(* CODESYS project SingleElevator_ancestor.project

Project tree, tasks and I/O mapping:
  Device : CODESYS Control Win V3, 3S - Smart Software Solutions GmbH, version 3.5.15.40
    application Application
      libraries: Standard, * (System)
      task MainTask (cyclic, interval 50 ms, priority 1) calls Simulation, GA_collector, Policy
      task VISU_TASK (cyclic, interval 100 ms, priority 31) calls VisuElems.Visu_Prg
      global variables GVL
      visualisation Visualization
      program Simulation [ST]
      GAs/
        function block Door_module [SFC]: ready_active, busy_active, op_complete_active, reset_done_active
        function block Dir_Vel_module [SFC]: go_fast_active, op_complete_active, reset_done_active, busy_active, ready_active, go_slow_active, stop_active
        function block Homing_Limit_module [SFC]: op_complete_active, reset_done_active, busy_active, ready_active, closing_doors_exit, closing_doors_active, slow_d_active, slow_u_active, opening_doors_active, opening_doors_exit, slow_u_top_active, slow_d_top_active, slow_d_exit, slow_u_exit, slow_u_top_exit, slow_d_top_exit, slow_d_bot_exit, slow_d_bot_exit_0, slow_u_bot_active, slow_d_bot_active, stop_h_active, stop_h_exit
        function block Calls_module [SFC]: Busy_active, Ready_active, op_complete_active, reset_done_active, save_up_active, Init_active, save_down_active, compose_array_up_active, compose_array_down_active
        function block Lights_module [SFC]: Ready_active, all_lights_active, Busy_active, save_call_active, save_call_exit
        function block Serve_call_module [SFC]: Ready_active, Busy_active, close_door_exit, slow_d_active, slow_d_exit, close_door_active, slow_u_active, fast_u_active, slow_u_land_active, Stop_active, Open_Doors_active, slow_u_exit, fast_u_exit, slow_u_land_exit, Stop_u_exit, Open_Doors_exit, fast_d_active, slow_d_land_active, Stop_d_active, fast_d_exit, slow_d_land_exit, Stop_d_exit, cancel_call_active, cancel_call_down_active, cancel_call_up_exit, cancel_call_down_exit
      program GA_collector [FBD]
      program Policy [SFC]: homing_active, homing_exit, wait_for_call_active
  text list GlobalTextList
*)

// Device/Application/GVL
//{attribute 'qualified_only'}
VAR_GLOBAL
(* Elevator managing variables*)
	Open: BOOL;				(* Sensor: the door is fully open*)
	Closed: BOOL;			(* Sensor: the door is fully closed*)
	LimitDown: BOOL;		(* Sensor: lower limit sensor, if TRUE the lift has reached the lower limit*)
	LimitUp: BOOL;			(* Sensor: upper limit sensor, if TRUE the lift has reached the upper limit*)
	DeckSensor: BOOL;		(* Sensor: if TRUE the cab is in proximity of a deck*)
	RampSensor: BOOL;		(* Sensor: if TRUE the cab is in proximity of a ramp*)
	Presence :BOOL; 		(* Sensor: if TRUE something blocks the door photocell*)
	Emergency: BOOL;		(* Input: if TRUE the emergency button has been pressed*)

	Closing: BOOL;			(* Actuator: if TRUE the door starts closing*)
	Opening: BOOL;			(* Actuator: the door starts opening*)
	Motor_on: BOOL;			(* Actuator: if TRUE the lift pulley motor start moving*)
	Up: BOOL;				(* Actuator parameter: if TRUE the lift moves upward, downward otherwise*)
	Vel: BOOL;				(* Actuator parameter: motor speed, if TRUE high speed, low speed otherwise*)
	

	Current: INT;  			(* Visualization: variable used to storage the current deck*)
    Destination: INT;		(* Visualization: variable used to storage the the destination deck*)
	EmergencyVis: BOOL; 	(* Visualization: if TRUE the emergency light is turned on*)

	
	
	
	
	
	InitialDeck: INT := 1;	(* Only for simulation: variable used to define the initial deck*)
	InitCycle: BOOL := FALSE;(* Only for simulation: used to execute the instruction at the first cycle*)
	Height: INT;			(* Only for simulation: elevator height*)
	DeckRest: INT;        	(* Only for simulation: division rest for generating deck sensor*)
	Memory: INT;
	RampRest: INT;			(* Only for simulation: division rest for generating the ramp position*)
	MemoryR: INT;
	Door: INT;				(* Only for simulation: to visualize the closing of the door*)
	Displacement: INT;		(* Only for simulation: lift displacement, dependent on the motor speed*)

 (*Inputs: internal panel variables*)
	PG: BOOL;
	P1: BOOL;
	P2: BOOL;
	P3: BOOL;
	P4: BOOL;
	P5: BOOL;
	P6: BOOL;
	P7: BOOL;

(*Visualization: internal panel variables used to turn on the LED*)
	PGVis: BOOL;
	P1Vis: BOOL;
	P2Vis: BOOL;
	P3Vis: BOOL;
	P4Vis: BOOL;
	P5Vis: BOOL;
	P6Vis: BOOL;
	P7Vis: BOOL;

(*Inputs: external panel variables*)
	UpDeckG: BOOL;
	UpDeck1: BOOL;
	UpDeck2: BOOL;
	UpDeck3: BOOL;
	UpDeck4: BOOL;
	UpDeck5: BOOL;
	UpDeck6: BOOL;
	DownDeck7: BOOL;
	DownDeck6: BOOL;
	DownDeck5: BOOL;
	DownDeck4: BOOL;
	DownDeck3: BOOL;
	DownDeck2: BOOL;
	DownDeck1: BOOL;

(*Visualization: external panel variables used to turn on the LED*)
	UpDeckGVis: BOOL;
	UpDeck1Vis: BOOL;
	UpDeck2Vis: BOOL;
	UpDeck3Vis: BOOL;
	UpDeck4Vis: BOOL;
	UpDeck5Vis: BOOL;
	UpDeck6Vis: BOOL;
	DownDeck7Vis: BOOL;
	DownDeck6Vis: BOOL;
	DownDeck5Vis: BOOL;
	DownDeck4Vis: BOOL;
	DownDeck3Vis: BOOL;
	DownDeck2Vis: BOOL;
	DownDeck1Vis: BOOL;

(*Only for simulation: variables used to simulate the fault on deck sensor*)
	SensorG: BOOL;				(* if TRUE the magnetic information for deck G is lost and the deck sensor cannot become TRUE*)
	Sensor1: BOOL;				(* if TRUE the magnetic information for deck 1 is lost and the deck sensor cannot become TRUE*)
	Sensor2: BOOL;
	Sensor3: BOOL;
	Sensor4: BOOL;
	Sensor5: BOOL;
	Sensor6: BOOL;
	Sensor7: BOOL;
	FaultSensorAlarm: BOOL; 	(* Visulaization: if TRUE alerts the user of a deck sensor fault*)

(*Only for simulation: variables used to simulate the fault on ramp sensor*)
	RampGUp: BOOL;
	Ramp1Down: BOOL;
	Ramp1Up:BOOL;
	Ramp2Down: BOOL;
	Ramp2Up:BOOL;
	Ramp3Down: BOOL;
	Ramp3Up:BOOL;
	Ramp4Down: BOOL;
	Ramp4Up:BOOL;
	Ramp5Down: BOOL;
	Ramp5Up:BOOL;
	Ramp6Down: BOOL;
	Ramp6Up:BOOL;
	Ramp7Down: BOOL;
	FaultRampAlarm: BOOL; 		(* Visulaization: if TRUE alerts the user of a ramp sensor fault*)
	SensorGOK: BOOL;
	Sensor1OK: BOOL;
	Sensor2OK: BOOL;
	Sensor6OK: BOOL;
	Sensor3OK: BOOL;
	Sensor4OK: BOOL;
	Sensor5OK: BOOL;
	Sensor7OK: BOOL;
	RampGUpOK: BOOL;
	Ramp1DownOK: BOOL;
	Ramp1UpOK: BOOL;
	Ramp2DownOK: BOOL;
	Ramp2UpOK: BOOL;
	Ramp3DownOK: BOOL;
	Ramp3UpOK: BOOL;
	Ramp4DownOK: BOOL;
	Ramp4UpOK: BOOL;
	Ramp5DownOK: BOOL;
	Ramp5UpOK: BOOL;
	Ramp6DownOK: BOOL;
	Ramp6UpOK: BOOL;
	Ramp7DownOK: BOOL;
	Ramp7UpOK: BOOL;
	//var aggiunte da me
	array_prio_up_onfly: ARRAY[0..7] OF INT;
	array_dest_up_onfly: ARRAY[0..7] OF INT;
	array_prio_up_stored: ARRAY[0..7] OF INT;
	array_dest_up_stored: ARRAY[0..7] OF INT;
	
	array_prio_down_onfly: ARRAY[0..7] OF INT;
	array_dest_down_onfly: ARRAY[0..7] OF INT;
	array_prio_down_stored: ARRAY[0..7] OF INT;
	array_dest_down_stored: ARRAY[0..7] OF INT;
	
	same_floor: BOOL; //flag di calls_module per la policy
	up_flag: BOOL; //
	RampSensor_target: BOOL;
	
	//Istanze dei GA
	door_module_0: Door_module;
	Dir_Vel_module_0: Dir_Vel_module;
	Homing_Limit_module_0: Homing_Limit_module;
	Lights_module_0: Lights_module;
	Calls_module_0: Calls_module;
	Serve_call_module_0: Serve_call_module;
	

END_VAR

// Device/Application/Simulation
PROGRAM Simulation
VAR
END_VAR

(* Initial position of the cab inside the hoistway. It is executed only at the first cycle.  *)
IF NOT GVL.InitCycle THEN
			GVL.InitCycle := TRUE ;
			GVL.Height := 20 * GVL.InitialDeck;
		    GVL.Door := 0;
			GVL.Current := GVL.Height / 20;
END_IF;

(* Elevator management, these instructions are executed each cycle time*)

(* Elevator door control. *)
IF GVL.Closing THEN
	GVL.Door := GVL.Door + 1;		(*Closing door management*)
	GVL.Open := FALSE;
END_IF

IF GVL.Door >= 60 THEN						(* Closed door limit*)
	GVL.Closed := TRUE;
END_IF

IF GVL.Opening THEN
	GVL.Door := GVL.Door - 1; 	(* Opening door management*)
	GVL.Closed := FALSE;
END_IF

IF GVL.Door <= 0 THEN							(* Open door limit*)
	GVL.Open := TRUE;
END_IF


(* Maximum and minimum management in the door simulation*)
IF GVL.Door < 0 THEN
	 GVL.Door := 0;
END_IF

IF GVL.Door > 60 THEN
	GVL.Door := 60;
END_IF


(* Control of the cab position inside the hostway. *)
(* Displacement definition for graphic visualization*)
IF GVL.Vel THEN 
	GVL.Displacement := 2;
ELSE 
	GVL.Displacement := 1;
END_IF


(* Height modification relying on direction and speed*)
IF GVL.Motor_on AND GVL.Up THEN
	GVL.Height := GVL.Height + GVL.Displacement;
	GVL.LimitDown := FALSE;
END_IF

IF GVL.Motor_on AND NOT GVL.Up THEN
	GVL.Height := GVL.Height - GVL.Displacement;
	GVL.LimitUp := FALSE;
END_IF


(* Limits for visualization*)
IF GVL.Height < -20 THEN
	GVL.Height := -20;
END_IF

IF GVL.Height > 160 THEN
	GVL.Height := 160;
END_IF

(* Limit sensors management*)
IF GVL.Height <= -10 THEN
	GVL.LimitDown := TRUE;
END_IF

IF GVL.Height >= 150 THEN
	 GVL.LimitUp := TRUE;
END_IF


(*-------------------------------------------------------------------*)
(*  Fault Management (Deck and Ramp Sensors)   *)
(*-------------------------------------------------------------------*)
(* Deck Sensor*)
(* Range of value where the deck sensor is active*)
IF ((GVL.Height >= -1) AND (GVL.Height <= 1)) THEN
	GVL.SensorGOK := TRUE;
ELSE  
	GVL.SensorGOK := FALSE;
END_IF

IF ((GVL.Height >= 20-1) AND (GVL.Height <= 20+1)) THEN
	GVL.Sensor1OK := TRUE;
ELSE  
	GVL.Sensor1OK := FALSE;
END_IF

IF ((GVL.Height >= 40-1) AND (GVL.Height <= 40+1)) THEN
	GVL.Sensor2OK := TRUE;
ELSE  
	GVL.Sensor2OK := FALSE;
END_IF

IF ((GVL.Height >= 60-1) AND (GVL.Height <= 60+1)) THEN
	GVL.Sensor3OK := TRUE;
ELSE  
	GVL.Sensor3OK := FALSE;
END_IF

IF ((GVL.Height >= 80-1) AND (GVL.Height <= 80+1)) THEN
	GVL.Sensor4OK := TRUE;
ELSE  
	GVL.Sensor4OK := FALSE;
END_IF

IF ((GVL.Height >= 100-1) AND (GVL.Height <= 100+1)) THEN
	GVL.Sensor5OK := TRUE;
ELSE   
	GVL.Sensor5OK := FALSE;
END_IF

IF ((GVL.Height >= 120-1) AND (GVL.Height <= 120+1)) THEN
	GVL.Sensor6OK := TRUE;
ELSE  
	GVL.Sensor6OK := FALSE;
END_IF

IF ((GVL.Height >= 140-1) AND (GVL.Height <= 140+1)) THEN
	GVL.Sensor7OK := TRUE;
ELSE  
	GVL.Sensor7OK := FALSE;
END_IF

GVL.DeckSensor := (GVL.SensorGOK AND NOT GVL.SensorG) OR
				    (GVL.Sensor1OK AND NOT GVL.Sensor1) OR
				    (GVL.Sensor2OK AND NOT GVL.Sensor2) OR
				    (GVL.Sensor3OK AND NOT GVL.Sensor3) OR
				    (GVL.Sensor4OK AND NOT GVL.Sensor4) OR
				    (GVL.Sensor5OK AND NOT GVL.Sensor5) OR
				    (GVL.Sensor6OK AND NOT GVL.Sensor6) OR
				    (GVL.Sensor7OK AND NOT GVL.Sensor7);

(* Ramp Sensor*)
(* Range of value where the ramp sensor is active*)
IF ((GVL.Height >= 5-1) AND (GVL.Height <= 5+1)) THEN
	GVL.RampGUpOK := TRUE;
ELSE 
	GVL.RampGUpOK := FALSE;
END_IF

(* Ramp close to deck 1*)
IF ((GVL.Height >= 15-1) AND (GVL.Height <= 15+1)) THEN
	GVL.Ramp1DownOK := TRUE;
ELSE 
	GVL.Ramp1DownOK := FALSE;
END_IF

IF ((GVL.Height >= 25-1) AND (GVL.Height <= 25+1)) THEN
	GVL.Ramp1UpOK := TRUE;
ELSE 
	GVL.Ramp1UpOK := FALSE;
END_IF

(* Ramp close to deck 2*)
IF ((GVL.Height >= 35-1) AND (GVL.Height <= 35+1)) THEN
	GVL.Ramp2DownOK := TRUE;
ELSE 
	GVL.Ramp2DownOK := FALSE;
END_IF

IF ((GVL.Height >= 45-1) AND (GVL.Height <= 45+1)) THEN
	GVL.Ramp2UpOK := TRUE;
ELSE 
	GVL.Ramp2UpOK := FALSE;
END_IF

(*Ramp close to deck  3*)
IF ((GVL.Height >= 55-1) AND (GVL.Height <= 55+1)) THEN
	GVL.Ramp3DownOK := TRUE;
ELSE 
	GVL.Ramp3DownOK := FALSE;
END_IF

IF ((GVL.Height >= 65-1) AND (GVL.Height <= 65+1)) THEN
	GVL.Ramp3UpOK := TRUE;
ELSE 
	GVL.Ramp3UpOK := FALSE;
END_IF

(* Ramp close to deck  4*)
IF ((GVL.Height >= 75-1) AND (GVL.Height <= 75+1)) THEN
	GVL.Ramp4DownOK := TRUE;
ELSE 
	GVL.Ramp4DownOK := FALSE;
END_IF

IF ((GVL.Height >= 85-1) AND (GVL.Height <= 85+1)) THEN
	GVL.Ramp4UpOK := TRUE;
ELSE 
	GVL.Ramp4UpOK:=FALSE;
END_IF

(* Ramp close to deck  5*)
IF ((GVL.Height >= 95-1) AND (GVL.Height <= 95+1)) THEN
	GVL.Ramp5DownOK := TRUE;
ELSE 
	GVL.Ramp5DownOK := FALSE;
END_IF

IF ((GVL.Height >= 105-1) AND (GVL.Height <= 105+1)) THEN
	GVL.Ramp5UpOK := TRUE;
ELSE
	GVL.Ramp5UpOK := FALSE;
END_IF

(* Ramp close to deck  6*)
IF ((GVL.Height >= 115-1) AND (GVL.Height <= 115+1)) THEN
	GVL.Ramp6DownOK := TRUE;
ELSE 
	GVL.Ramp6DownOK := FALSE;
END_IF

IF ((GVL.Height >= 125-1) AND (GVL.Height <= 125+1)) THEN
	GVL.Ramp6UpOK := TRUE;
ELSE 
	GVL.Ramp6UpOK := FALSE;
END_IF

(* Ramp close to deck  7*)
IF ((GVL.Height >= 135-1) AND (GVL.Height <= 135+1)) THEN
	GVL.Ramp7DownOK := TRUE;
ELSE 
	GVL.Ramp7DownOK := FALSE;
END_IF

GVL.RampSensor:=(GVL.RampGUpOK AND NOT GVL.RampGUp) OR 
								(GVL.Ramp1DownOK AND NOT GVL.Ramp1Down ) OR 
								(GVL.Ramp1UpOK AND NOT GVL.Ramp1Up ) OR
								(GVL.Ramp2DownOK AND NOT GVL.Ramp2Down ) OR 
								(GVL.Ramp2UpOK AND NOT GVL.Ramp2Up ) OR
								(GVL.Ramp3DownOK AND NOT GVL.Ramp3Down ) OR
 								(GVL.Ramp3UpOK AND NOT GVL.Ramp3Up ) OR
								(GVL.Ramp4DownOK AND NOT GVL.Ramp4Down ) OR
 								(GVL.Ramp4UpOK AND NOT GVL.Ramp4Up ) OR
								(GVL.Ramp5DownOK AND NOT GVL.Ramp5Down ) OR
 								(GVL.Ramp5UpOK AND NOT GVL.Ramp5Up ) OR
								(GVL.Ramp6DownOK AND NOT GVL.Ramp6Down ) OR
								(GVL.Ramp6UpOK AND NOT GVL.Ramp6Up ) OR
								(GVL.Ramp7DownOK AND NOT GVL.Ramp7Down );

END_PROGRAM

// Device/Application/GA_collector
PROGRAM GA_collector
VAR


END_VAR

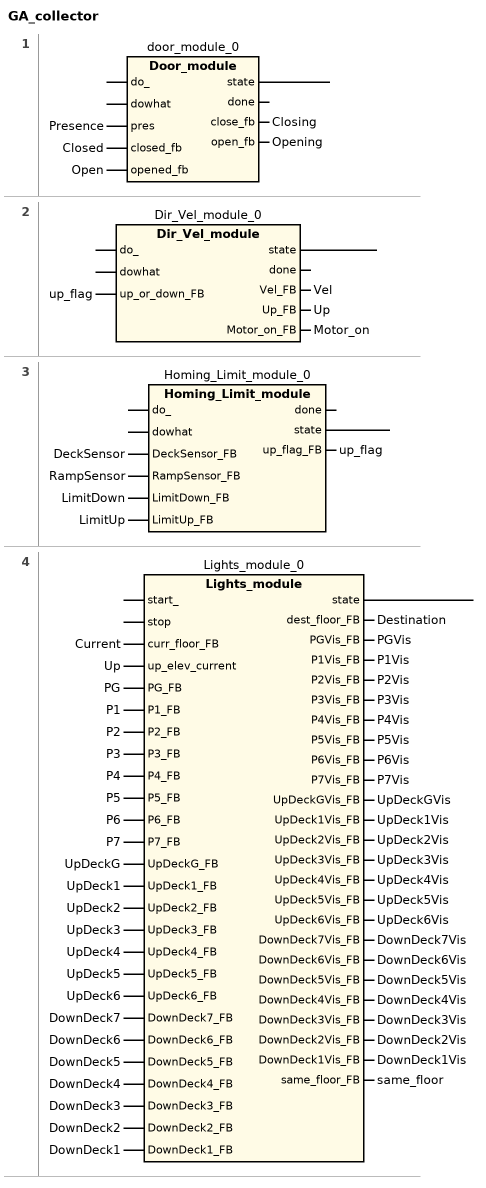
// NETWORK 1
door_module_0(
    pres := Presence,
    closed_fb := Closed,
    opened_fb := Open,
    close_fb => Closing,
    open_fb => Opening); // Door_module

// NETWORK 2
Dir_Vel_module_0(up_or_down_FB := up_flag, Vel_FB => Vel, Up_FB => Up, Motor_on_FB => Motor_on); // Dir_Vel_module

// NETWORK 3
Homing_Limit_module_0(
    DeckSensor_FB := DeckSensor,
    RampSensor_FB := RampSensor,
    LimitDown_FB := LimitDown,
    LimitUp_FB := LimitUp,
    up_flag_FB => up_flag); // Homing_Limit_module

// NETWORK 4
Lights_module_0(
    curr_floor_FB := Current,
    up_elev_current := Up,
    PG_FB := PG,
    P1_FB := P1,
    P2_FB := P2,
    P3_FB := P3,
    P4_FB := P4,
    P5_FB := P5,
    P6_FB := P6,
    P7_FB := P7,
    UpDeckG_FB := UpDeckG,
    UpDeck1_FB := UpDeck1,
    UpDeck2_FB := UpDeck2,
    UpDeck3_FB := UpDeck3,
    UpDeck4_FB := UpDeck4,
    UpDeck5_FB := UpDeck5,
    UpDeck6_FB := UpDeck6,
    DownDeck7_FB := DownDeck7,
    DownDeck6_FB := DownDeck6,
    DownDeck5_FB := DownDeck5,
    DownDeck4_FB := DownDeck4,
    DownDeck3_FB := DownDeck3,
    DownDeck2_FB := DownDeck2,
    DownDeck1_FB := DownDeck1,
    dest_floor_FB => Destination,
    PGVis_FB => PGVis,
    P1Vis_FB => P1Vis,
    P2Vis_FB => P2Vis,
    P3Vis_FB => P3Vis,
    P4Vis_FB => P4Vis,
    P5Vis_FB => P5Vis,
    P6Vis_FB => P6Vis,
    P7Vis_FB => P7Vis,
    UpDeckGVis_FB => UpDeckGVis,
    UpDeck1Vis_FB => UpDeck1Vis,
    UpDeck2Vis_FB => UpDeck2Vis,
    UpDeck3Vis_FB => UpDeck3Vis,
    UpDeck4Vis_FB => UpDeck4Vis,
    UpDeck5Vis_FB => UpDeck5Vis,
    UpDeck6Vis_FB => UpDeck6Vis,
    DownDeck7Vis_FB => DownDeck7Vis,
    DownDeck6Vis_FB => DownDeck6Vis,
    DownDeck5Vis_FB => DownDeck5Vis,
    DownDeck4Vis_FB => DownDeck4Vis,
    DownDeck3Vis_FB => DownDeck3Vis,
    DownDeck2Vis_FB => DownDeck2Vis,
    DownDeck1Vis_FB => DownDeck1Vis,
    same_floor_FB => same_floor); // Lights_module

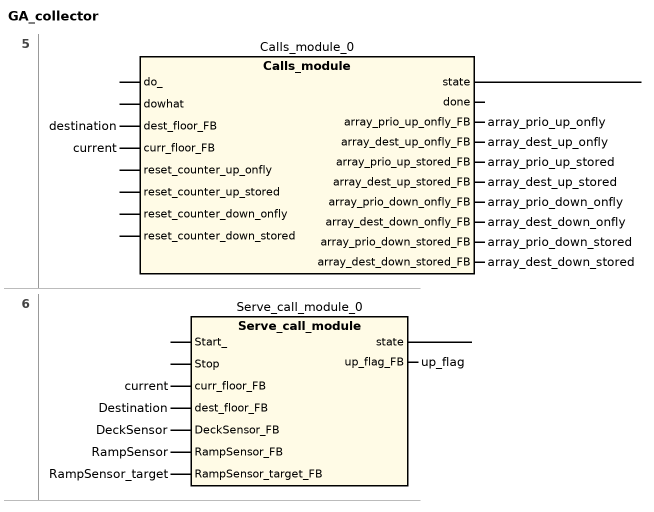
// NETWORK 5
Calls_module_0(
    dest_floor_FB := destination,
    curr_floor_FB := current,
    array_prio_up_onfly_FB => array_prio_up_onfly,
    array_dest_up_onfly_FB => array_dest_up_onfly,
    array_prio_up_stored_FB => array_prio_up_stored,
    array_dest_up_stored_FB => array_dest_up_stored,
    array_prio_down_onfly_FB => array_prio_down_onfly,
    array_dest_down_onfly_FB => array_dest_down_onfly,
    array_prio_down_stored_FB => array_prio_down_stored,
    array_dest_down_stored_FB => array_dest_down_stored); // Calls_module

// NETWORK 6
Serve_call_module_0(
    curr_floor_FB := current,
    dest_floor_FB := Destination,
    DeckSensor_FB := DeckSensor,
    RampSensor_FB := RampSensor,
    RampSensor_target_FB := RampSensor_target,
    up_flag_FB => up_flag); // Serve_call_module

END_PROGRAM

// Device/Application/GAs/Door_module
FUNCTION_BLOCK Door_module
VAR_INPUT
	do_: BOOL;
	dowhat: STRING;
	pres: BOOL;
	closed_fb: BOOL;
	opened_fb: BOOL;
END_VAR
VAR_OUTPUT
	state: STRING;
	done: BOOL;
	close_fb: BOOL;
	open_fb: BOOL;
END_VAR
VAR
END_VAR

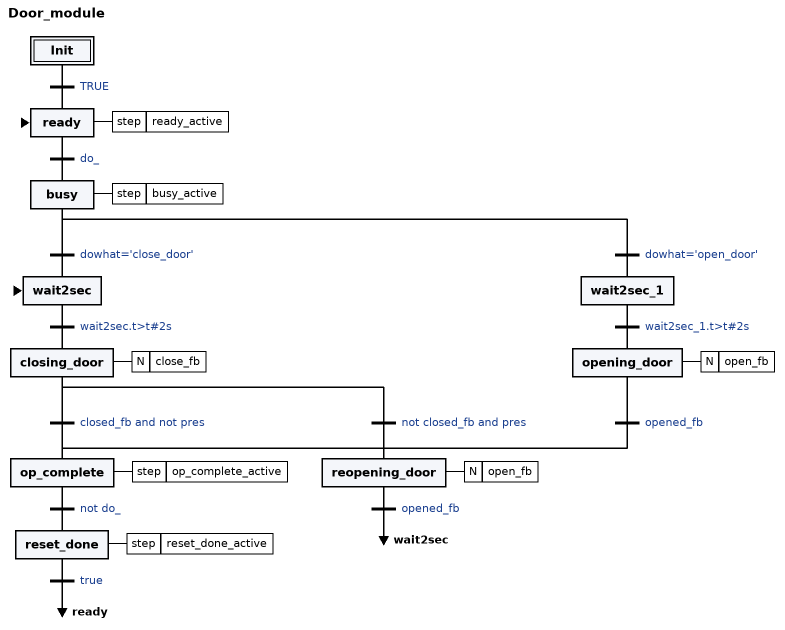
INITIAL_STEP Init:
END_STEP
TRANSITION FROM Init TO ready
    := TRUE;
END_TRANSITION
STEP ready:
    ready_active(N);  // step action
END_STEP
TRANSITION FROM ready TO busy
    := do_;
END_TRANSITION
STEP busy:
    busy_active(N);  // step action
END_STEP
TRANSITION FROM busy TO wait2sec
    := dowhat='close_door';
END_TRANSITION
STEP wait2sec:
END_STEP
TRANSITION FROM wait2sec TO closing_door
    := wait2sec.t>t#2s;
END_TRANSITION
STEP closing_door:
    close_fb(N);
END_STEP
TRANSITION FROM closing_door TO op_complete
    := closed_fb and not pres;
END_TRANSITION
TRANSITION FROM closing_door TO reopening_door
    := not closed_fb and pres;
END_TRANSITION
STEP reopening_door:
    open_fb(N);
END_STEP
TRANSITION FROM reopening_door TO wait2sec
    := opened_fb;
END_TRANSITION
TRANSITION FROM busy TO wait2sec_1
    := dowhat='open_door';
END_TRANSITION
STEP wait2sec_1:
END_STEP
TRANSITION FROM wait2sec_1 TO opening_door
    := wait2sec_1.t>t#2s;
END_TRANSITION
STEP opening_door:
    open_fb(N);
END_STEP
TRANSITION FROM opening_door TO op_complete
    := opened_fb;
END_TRANSITION
STEP op_complete:
    op_complete_active(N);  // step action
END_STEP
TRANSITION FROM op_complete TO reset_done
    := not do_;
END_TRANSITION
STEP reset_done:
    reset_done_active(N);  // step action
END_STEP
TRANSITION FROM reset_done TO ready
    := true;
END_TRANSITION

ACTION ready_active:
state:='Ready';
END_ACTION

ACTION busy_active:
state:='Busy';
END_ACTION

ACTION op_complete_active:
done:=TRUE;
END_ACTION

ACTION reset_done_active:
done:=FALSE;
END_ACTION

END_FUNCTION_BLOCK

// Device/Application/GAs/Dir_Vel_module
FUNCTION_BLOCK Dir_Vel_module
VAR_INPUT
	do_: BOOL;
	dowhat: STRING;
	up_or_down_FB: BOOL;
END_VAR
VAR_OUTPUT
	state: STRING;
	done: BOOL;
	Vel_FB: BOOL;
	Up_FB: BOOL;
	Motor_on_FB: BOOL;
END_VAR
VAR
END_VAR

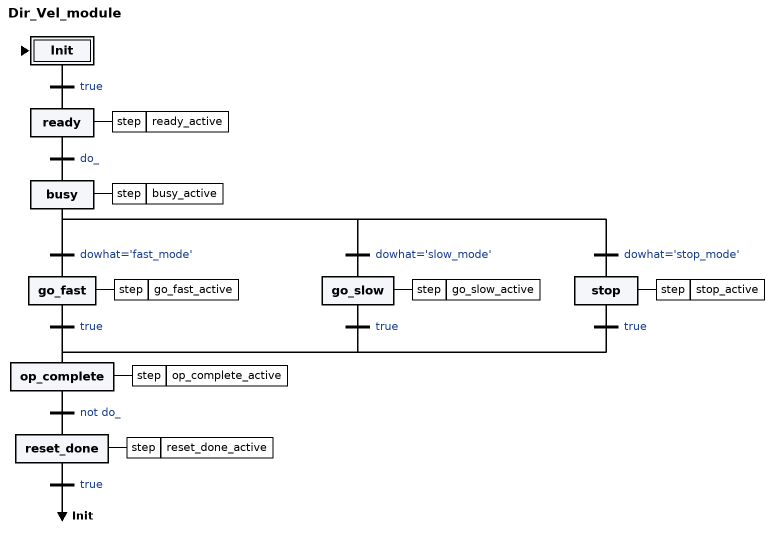
INITIAL_STEP Init:
END_STEP
TRANSITION FROM Init TO ready
    := true;
END_TRANSITION
STEP ready:
    ready_active(N);  // step action
END_STEP
TRANSITION FROM ready TO busy
    := do_;
END_TRANSITION
STEP busy:
    busy_active(N);  // step action
END_STEP
TRANSITION FROM busy TO go_fast
    := dowhat='fast_mode';
END_TRANSITION
STEP go_fast:
    go_fast_active(N);  // step action
END_STEP
TRANSITION FROM go_fast TO op_complete
    := true;
END_TRANSITION
TRANSITION FROM busy TO go_slow
    := dowhat='slow_mode';
END_TRANSITION
STEP go_slow:
    go_slow_active(N);  // step action
END_STEP
TRANSITION FROM go_slow TO op_complete
    := true;
END_TRANSITION
TRANSITION FROM busy TO stop
    := dowhat='stop_mode';
END_TRANSITION
STEP stop:
    stop_active(N);  // step action
END_STEP
TRANSITION FROM stop TO op_complete
    := true;
END_TRANSITION
STEP op_complete:
    op_complete_active(N);  // step action
END_STEP
TRANSITION FROM op_complete TO reset_done
    := not do_;
END_TRANSITION
STEP reset_done:
    reset_done_active(N);  // step action
END_STEP
TRANSITION FROM reset_done TO Init
    := true;
END_TRANSITION

ACTION go_fast_active:
Motor_on_FB:= TRUE;
Vel_FB:= TRUE;
END_ACTION

ACTION op_complete_active:
done:=TRUE;
END_ACTION

ACTION reset_done_active:
done:=FALSE;
END_ACTION

ACTION busy_active:
state:='Busy';
IF  up_or_down_FB THEN
	Up_FB:=TRUE;
ELSE
	Up_FB:=FALSE;
END_IF
END_ACTION

ACTION ready_active:
state:='Ready';
END_ACTION

ACTION go_slow_active:
Motor_on_FB:= TRUE;
Vel_FB:= FALSE;
END_ACTION

ACTION stop_active:
Motor_on_FB:= FALSE;
END_ACTION

END_FUNCTION_BLOCK

// Device/Application/GAs/Homing_Limit_module
FUNCTION_BLOCK Homing_Limit_module
VAR_INPUT
	do_: BOOL;
	dowhat: STRING;
	DeckSensor_FB: BOOL;
	RampSensor_FB: BOOL;
	LimitDown_FB: BOOL;
	LimitUp_FB: BOOL;
END_VAR
VAR_OUTPUT
	done: BOOL;
	state: STRING;
	up_flag_FB: BOOL;
END_VAR
VAR
	sync: BOOL;
	Opok: BOOL;
END_VAR

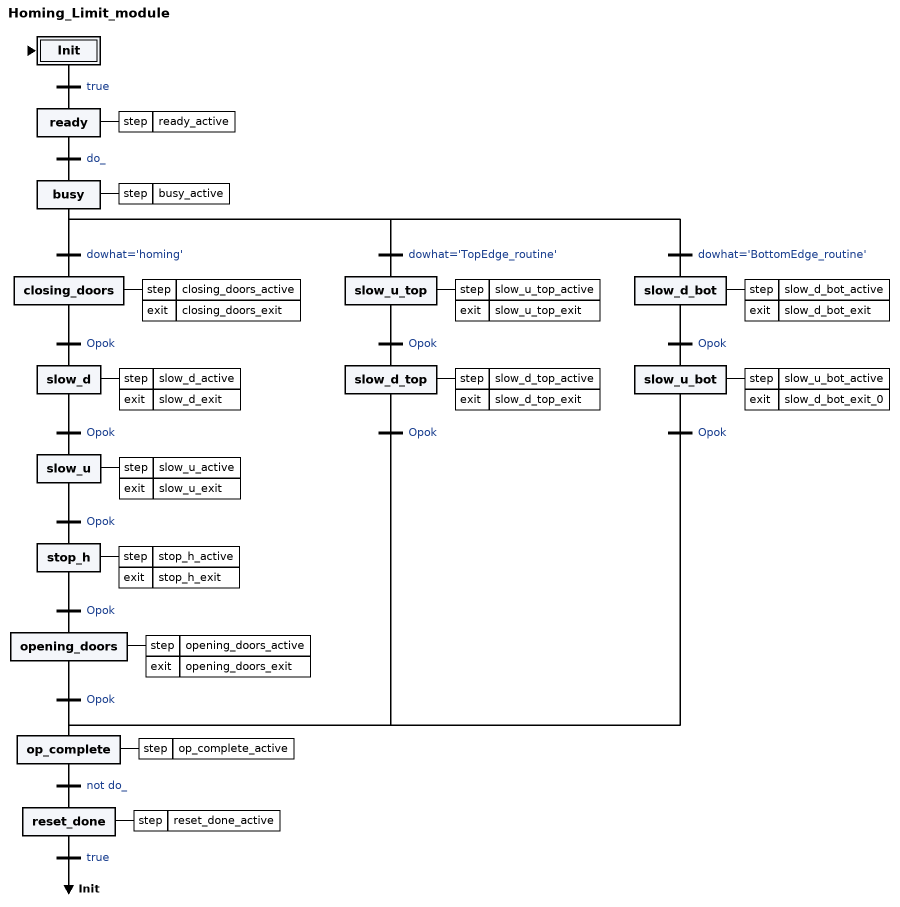
INITIAL_STEP Init:
END_STEP
TRANSITION FROM Init TO ready
    := true;
END_TRANSITION
STEP ready:
    ready_active(N);  // step action
END_STEP
TRANSITION FROM ready TO busy
    := do_;
END_TRANSITION
STEP busy:
    busy_active(N);  // step action
END_STEP
TRANSITION FROM busy TO closing_doors
    := dowhat='homing';
END_TRANSITION
STEP closing_doors:
    closing_doors_active(N);  // step action
    closing_doors_exit(P0);  // exit action
END_STEP
TRANSITION FROM closing_doors TO slow_d
    := Opok;
END_TRANSITION
STEP slow_d:
    slow_d_active(N);  // step action
    slow_d_exit(P0);  // exit action
END_STEP
TRANSITION FROM slow_d TO slow_u
    := Opok;
END_TRANSITION
STEP slow_u:
    slow_u_active(N);  // step action
    slow_u_exit(P0);  // exit action
END_STEP
TRANSITION FROM slow_u TO stop_h
    := Opok;
END_TRANSITION
STEP stop_h:
    stop_h_active(N);  // step action
    stop_h_exit(P0);  // exit action
END_STEP
TRANSITION FROM stop_h TO opening_doors
    := Opok;
END_TRANSITION
STEP opening_doors:
    opening_doors_active(N);  // step action
    opening_doors_exit(P0);  // exit action
END_STEP
TRANSITION FROM opening_doors TO op_complete
    := Opok;
END_TRANSITION
TRANSITION FROM busy TO slow_u_top
    := dowhat='TopEdge_routine';
END_TRANSITION
STEP slow_u_top:
    slow_u_top_active(N);  // step action
    slow_u_top_exit(P0);  // exit action
END_STEP
TRANSITION FROM slow_u_top TO slow_d_top
    := Opok;
END_TRANSITION
STEP slow_d_top:
    slow_d_top_active(N);  // step action
    slow_d_top_exit(P0);  // exit action
END_STEP
TRANSITION FROM slow_d_top TO op_complete
    := Opok;
END_TRANSITION
TRANSITION FROM busy TO slow_d_bot
    := dowhat='BottomEdge_routine';
END_TRANSITION
STEP slow_d_bot:
    slow_d_bot_active(N);  // step action
    slow_d_bot_exit(P0);  // exit action
END_STEP
TRANSITION FROM slow_d_bot TO slow_u_bot
    := Opok;
END_TRANSITION
STEP slow_u_bot:
    slow_u_bot_active(N);  // step action
    slow_d_bot_exit_0(P0);  // exit action
END_STEP
TRANSITION FROM slow_u_bot TO op_complete
    := Opok;
END_TRANSITION
STEP op_complete:
    op_complete_active(N);  // step action
END_STEP
TRANSITION FROM op_complete TO reset_done
    := not do_;
END_TRANSITION
STEP reset_done:
    reset_done_active(N);  // step action
END_STEP
TRANSITION FROM reset_done TO Init
    := true;
END_TRANSITION

ACTION op_complete_active:
done:=TRUE;
END_ACTION

ACTION reset_done_active:
done:=FALSE;
END_ACTION

ACTION busy_active:
state:='Busy';
END_ACTION

ACTION ready_active:
state:='Ready';
END_ACTION

ACTION closing_doors_exit:
sync:=FALSE;
Opok:=FALSE;
END_ACTION

ACTION closing_doors_active:
//CHIUSURA PORTE 
IF door_module_0.State='Ready' THEN
	door_module_0.Do_:=TRUE;
	door_module_0.DoWhat:='close_door';
END_IF

IF door_module_0.Done AND door_module_0.State='Busy' THEN
	door_module_0.Do_:=FALSE;
	sync:=TRUE;
END_IF

Opok:= sync and not door_module_0.Done;
END_ACTION

ACTION slow_d_active:
//DISCESA VERSO IL BASSO
IF Dir_Vel_module_0.State='Ready' THEN
	Dir_Vel_module_0.Do_:=TRUE;
	Dir_Vel_module_0.DoWhat:='slow_mode';
	up_flag_FB:=FALSE;
END_IF

IF Dir_Vel_module_0.Done AND Dir_Vel_module_0.State='Busy' AND LimitDown_FB THEN
	Dir_Vel_module_0.Do_:=FALSE;
	sync:=TRUE;
END_IF

Opok:= sync AND NOT Dir_Vel_module_0.Done;
END_ACTION

ACTION slow_u_active:
//SALITA VERSO L'ALTO
IF Dir_Vel_module_0.State='Ready' THEN
	Dir_Vel_module_0.Do_:=TRUE;
	Dir_Vel_module_0.DoWhat:='slow_mode';
	up_flag_FB:=TRUE;
END_IF

IF Dir_Vel_module_0.Done AND Dir_Vel_module_0.State='Busy' AND DeckSensor_FB THEN
	Dir_Vel_module_0.Do_:=FALSE;
	sync:=TRUE;
END_IF

Opok:= sync AND NOT Dir_Vel_module_0.Done;
END_ACTION

ACTION opening_doors_active:
//APERTURA PORTE 
IF door_module_0.State='Ready' THEN
	door_module_0.Do_:=TRUE;
	door_module_0.DoWhat:='open_door';
END_IF

IF door_module_0.Done AND door_module_0.State='Busy' THEN
	door_module_0.Do_:=FALSE;
	sync:=TRUE;
END_IF

Opok:= sync AND NOT door_module_0.Done;
END_ACTION

ACTION opening_doors_exit:
sync:=FALSE;
Opok:=FALSE;
END_ACTION

ACTION slow_u_top_active:
//SALITA VERSO L'ALTO LENTA
IF Dir_Vel_module_0.State='Ready' THEN
	Dir_Vel_module_0.Do_:=TRUE;
	Dir_Vel_module_0.DoWhat:='slow_mode';
	up_flag_FB:=TRUE;
END_IF

IF Dir_Vel_module_0.Done AND Dir_Vel_module_0.State='Busy' AND LimitUp_FB THEN
	Dir_Vel_module_0.Do_:=FALSE;
	sync:=TRUE;
END_IF

Opok:= sync AND NOT Dir_Vel_module_0.Done;
END_ACTION

ACTION slow_d_top_active:
//DISCESA VERSO IL BASSO LENTA
IF Dir_Vel_module_0.State='Ready' THEN
	Dir_Vel_module_0.Do_:=TRUE;
	Dir_Vel_module_0.DoWhat:='slow_mode';
	up_flag_FB:=FALSE;
END_IF

IF Dir_Vel_module_0.Done AND Dir_Vel_module_0.State='Busy' AND RampSensor_FB THEN
	Dir_Vel_module_0.Do_:=FALSE;
	sync:=TRUE;
END_IF

Opok:= sync AND NOT Dir_Vel_module_0.Done;
END_ACTION

ACTION slow_d_exit:
sync:=FALSE;
Opok:=FALSE;
END_ACTION

ACTION slow_u_exit:
sync:=FALSE;
Opok:=FALSE;
END_ACTION

ACTION slow_u_top_exit:
sync:=FALSE;
Opok:=FALSE;
END_ACTION

ACTION slow_d_top_exit:
sync:=FALSE;
Opok:=FALSE;
END_ACTION

ACTION slow_d_bot_exit:
sync:=FALSE;
Opok:=FALSE;
END_ACTION

ACTION slow_d_bot_exit_0:
sync:=FALSE;
Opok:=FALSE;
END_ACTION

ACTION slow_u_bot_active:
//SALITA VERSO L'ALTO LENTA
IF Dir_Vel_module_0.State='Ready' THEN
	Dir_Vel_module_0.Do_:=TRUE;
	Dir_Vel_module_0.DoWhat:='slow_mode';
	up_flag_FB:=TRUE;
END_IF

IF Dir_Vel_module_0.Done AND Dir_Vel_module_0.State='Busy' AND RampSensor_FB THEN
	Dir_Vel_module_0.Do_:=FALSE;
	sync:=TRUE;
END_IF

Opok:= sync AND NOT Dir_Vel_module_0.Done;
END_ACTION

ACTION slow_d_bot_active:
//DISCESA VERSO IL BASSO LENTA
IF Dir_Vel_module_0.State='Ready' THEN
	Dir_Vel_module_0.Do_:=TRUE;
	Dir_Vel_module_0.DoWhat:='slow_mode';
	up_flag_FB:=FALSE;
END_IF

IF Dir_Vel_module_0.Done AND Dir_Vel_module_0.State='Busy' AND LimitDown_FB THEN
	Dir_Vel_module_0.Do_:=FALSE;
	sync:=TRUE;
END_IF

Opok:= sync AND NOT Dir_Vel_module_0.Done;
END_ACTION

ACTION stop_h_active:
//STOP
IF Dir_Vel_module_0.State='Ready' THEN
	Dir_Vel_module_0.Do_:=TRUE;
	Dir_Vel_module_0.DoWhat:='stop_mode';
END_IF

IF Dir_Vel_module_0.Done AND Dir_Vel_module_0.State='Busy' THEN
	Dir_Vel_module_0.Do_:=FALSE;
	sync:=TRUE;
END_IF

Opok:= sync AND NOT Dir_Vel_module_0.Done;
END_ACTION

ACTION stop_h_exit:
sync:=FALSE;
Opok:=FALSE;
END_ACTION

END_FUNCTION_BLOCK

// Device/Application/GAs/Lights_module
FUNCTION_BLOCK Lights_module
VAR_INPUT
	start_: BOOL;
	stop: BOOL;

	curr_floor_FB: INT; //piano corrente
	up_elev_current:BOOL; //verso attuale di marcia
	(*Inputs: internal panel variables*)	
	PG_FB: BOOL;
	P1_FB: BOOL;
	P2_FB: BOOL;
	P3_FB: BOOL;
	P4_FB: BOOL;
	P5_FB: BOOL;
	P6_FB: BOOL;
	P7_FB: BOOL;
	(*Inputs: external panel variables*)
	UpDeckG_FB: BOOL;
	UpDeck1_FB: BOOL;
	UpDeck2_FB: BOOL;
	UpDeck3_FB: BOOL;
	UpDeck4_FB: BOOL;
	UpDeck5_FB: BOOL;
	UpDeck6_FB: BOOL;
	DownDeck7_FB: BOOL;
	DownDeck6_FB: BOOL;
	DownDeck5_FB: BOOL;
	DownDeck4_FB: BOOL;
	DownDeck3_FB: BOOL;
	DownDeck2_FB: BOOL;
	DownDeck1_FB: BOOL;

END_VAR
VAR_OUTPUT
	state: STRING;
	dest_floor_FB: INT; //piano di destinazione 
	(*Visualization: internal panel variables used TO turn on the LED*)
	PGVis_FB: BOOL;
	P1Vis_FB: BOOL;
	P2Vis_FB: BOOL;
	P3Vis_FB: BOOL;
	P4Vis_FB: BOOL;
	P5Vis_FB: BOOL;
	P6Vis_FB: BOOL;
	P7Vis_FB: BOOL;
	(*Visualization: external panel variables used to turn on the LED*)
	UpDeckGVis_FB: BOOL;
	UpDeck1Vis_FB: BOOL;
	UpDeck2Vis_FB: BOOL;
	UpDeck3Vis_FB: BOOL;
	UpDeck4Vis_FB: BOOL;
	UpDeck5Vis_FB: BOOL;
	UpDeck6Vis_FB: BOOL;
	DownDeck7Vis_FB: BOOL;
	DownDeck6Vis_FB: BOOL;
	DownDeck5Vis_FB: BOOL;
	DownDeck4Vis_FB: BOOL;
	DownDeck3Vis_FB: BOOL;
	DownDeck2Vis_FB: BOOL;
	DownDeck1Vis_FB: BOOL;
	

	same_floor_FB: BOOL;
END_VAR
VAR
	up_motion_FB: BOOL; //verso della chiamata
	can_be_clicked: BOOL; //per non scrivere sulla var di Stop
	sync: BOOL;
	Opok: BOOL;
	contup: INT;
	reset_down_counter: BOOL;
END_VAR

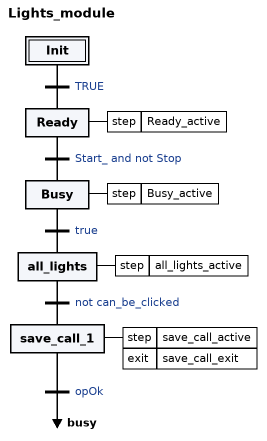
INITIAL_STEP Init:
END_STEP
TRANSITION FROM Init TO Ready
    := TRUE;
END_TRANSITION
STEP Ready:
    Ready_active(N);  // step action
END_STEP
TRANSITION FROM Ready TO Busy
    := Start_ and not Stop;
END_TRANSITION
STEP Busy:
    Busy_active(N);  // step action
END_STEP
TRANSITION FROM Busy TO all_lights
    := true;
END_TRANSITION
STEP all_lights:
    all_lights_active(N);  // step action
END_STEP
TRANSITION FROM all_lights TO save_call_1
    := not can_be_clicked;
END_TRANSITION
STEP save_call_1:
    save_call_active(N);  // step action
    save_call_exit(P0);  // exit action
END_STEP
TRANSITION FROM save_call_1 TO busy
    := opOk;
END_TRANSITION

ACTION Ready_active:
State:='ready';
END_ACTION

ACTION all_lights_active:
IF PG_FB AND can_be_clicked THEN
	PGVis_FB:=TRUE;
	can_be_clicked:=FALSE;
	dest_floor_FB:=0;
	up_motion_FB:= up_elev_current; // la chiamata ha verso pari al verso corrente dell'ascensore
END_IF
IF P1_FB AND can_be_clicked THEN
	P1Vis_FB:=TRUE;
	can_be_clicked:=FALSE;
	dest_floor_FB:=1;
	up_motion_FB:= up_elev_current;
END_IF
IF P2_FB AND can_be_clicked THEN
	P2Vis_FB:=TRUE;
	can_be_clicked:=FALSE;
	dest_floor_FB:=2;
	up_motion_FB:= up_elev_current;
END_IF
IF P3_FB AND can_be_clicked THEN
	P3Vis_FB:=TRUE;
	can_be_clicked:=FALSE;
	dest_floor_FB:=3;
	up_motion_FB:= up_elev_current;
END_IF
IF P4_FB AND can_be_clicked THEN
	P4Vis_FB:=TRUE;
	can_be_clicked:=FALSE;
	dest_floor_FB:=4;
	up_motion_FB:= up_elev_current;
END_IF
IF P5_FB AND can_be_clicked THEN
	P5Vis_FB:=TRUE;
	can_be_clicked:=FALSE;
	dest_floor_FB:=5;
	up_motion_FB:= up_elev_current;
END_IF
IF P6_FB AND can_be_clicked THEN
	P6Vis_FB:=TRUE;
	can_be_clicked:=FALSE;
	dest_floor_FB:=6;
	up_motion_FB:= up_elev_current;
END_IF
IF P7_FB AND can_be_clicked THEN
	P7Vis_FB:=TRUE;
	can_be_clicked:=FALSE;
	dest_floor_FB:=7;
	up_motion_FB:= up_elev_current;
END_IF

//luci esterne

IF UpDeckG_FB AND can_be_clicked THEN
	UpDeckGVis_FB:=TRUE;
	can_be_clicked:=FALSE;
	dest_floor_FB:=0;
	up_motion_FB:=TRUE;
END_IF
IF UpDeck1_FB AND can_be_clicked THEN
	UpDeck1Vis_FB:=TRUE;
	can_be_clicked:=FALSE;
	dest_floor_FB:=1;
	up_motion_FB:=TRUE;
END_IF
IF UpDeck2_FB AND can_be_clicked THEN
	UpDeck2Vis_FB:=TRUE;
	can_be_clicked:=FALSE;
	dest_floor_FB:=2;
	up_motion_FB:=TRUE;
END_IF
IF UpDeck3_FB AND can_be_clicked THEN
	UpDeck3Vis_FB:=TRUE;
	can_be_clicked:=FALSE;
	dest_floor_FB:=3;
	up_motion_FB:=TRUE;
END_IF
IF UpDeck4_FB AND can_be_clicked THEN
	UpDeck4Vis_FB:=TRUE;
	can_be_clicked:=FALSE;
	dest_floor_FB:=4;
	up_motion_FB:=TRUE;
END_IF
IF UpDeck5_FB AND can_be_clicked THEN
	UpDeck5Vis_FB:=TRUE;
	can_be_clicked:=FALSE;
	dest_floor_FB:=5;
	up_motion_FB:=TRUE;
END_IF
IF UpDeck6_FB AND can_be_clicked THEN
	UpDeck6Vis_FB:=TRUE;
	can_be_clicked:=FALSE;
	dest_floor_FB:=6;
	up_motion_FB:=TRUE;
END_IF
IF DownDeck7_FB AND can_be_clicked THEN
	DownDeck7Vis_FB:=TRUE;
	can_be_clicked:=FALSE;
	dest_floor_FB:=7;
	up_motion_FB:=FALSE;
END_IF
IF DownDeck6_FB AND can_be_clicked THEN
	DownDeck6Vis_FB:=TRUE;
	can_be_clicked:=FALSE;
	dest_floor_FB:=6;
	up_motion_FB:=FALSE;
END_IF
IF DownDeck5_FB AND can_be_clicked THEN
	DownDeck5Vis_FB:=TRUE;
	can_be_clicked:=FALSE;
	dest_floor_FB:=5;
	up_motion_FB:=FALSE;
END_IF
IF DownDeck4_FB AND can_be_clicked THEN
	DownDeck4Vis_FB:=TRUE;
	can_be_clicked:=FALSE;
	dest_floor_FB:=4;
	up_motion_FB:=FALSE;
END_IF
IF DownDeck3_FB AND can_be_clicked THEN
	DownDeck3Vis_FB:=TRUE;
	can_be_clicked:=FALSE;
	dest_floor_FB:=3;
	up_motion_FB:=FALSE;
END_IF
IF DownDeck2_FB AND can_be_clicked THEN
	DownDeck2Vis_FB:=TRUE;
	can_be_clicked:=FALSE;
	dest_floor_FB:=2;
	up_motion_FB:=FALSE;
END_IF
IF DownDeck1_FB AND can_be_clicked THEN
	DownDeck1Vis_FB:=TRUE;
	can_be_clicked:=FALSE;
	dest_floor_FB:=1;
	up_motion_FB:=FALSE;
END_IF
END_ACTION

ACTION Busy_active:
State:='busy';
can_be_clicked:=TRUE;
END_ACTION

ACTION save_call_active:
IF up_motion_FB THEN
//chiama calls per salvare su array calls_up	
	IF Calls_module_0.State='Ready' THEN
	Calls_module_0.Do_:=TRUE;
	Calls_module_0.DoWhat:='calls_up';
	END_IF

	IF Calls_module_0.Done AND Calls_module_0.State='Busy' THEN
		Calls_module_0.Do_:=FALSE;
		sync:=TRUE;
		contup:=contup+1;
	END_IF

	Opok:= sync AND NOT Calls_module_0.Done;
ELSE 

//chiama calls per salvare su array calls_down	
	IF Calls_module_0.State='Ready' THEN
	Calls_module_0.Do_:=TRUE;
	Calls_module_0.DoWhat:='calls_down';
	END_IF

	IF Calls_module_0.Done AND Calls_module_0.State='Busy' THEN
		Calls_module_0.Do_:=FALSE;
		sync:=TRUE;
	END_IF

	Opok:= sync AND NOT Calls_module_0.Done;
END_IF 

// SE LA CHIAMATA è SULLO STESSO FLOOR IN CUI STO ANDANDO
IF dest_floor_FB = curr_floor_FB THEN
	same_floor_FB:=TRUE;
ELSE
	same_floor_FB:=FALSE;
END_IF
END_ACTION

ACTION save_call_exit:
sync:=FALSE;
Opok:=FALSE;
END_ACTION

END_FUNCTION_BLOCK

// Device/Application/GAs/Calls_module
FUNCTION_BLOCK Calls_module
VAR_INPUT
	do_: BOOL;
	dowhat: STRING;
	dest_floor_FB: INT; //collegato a dest_floor
	curr_floor_FB: INT; //collegato a current della policy
END_VAR
VAR_OUTPUT
	state: STRING;
	done: BOOL;
	array_prio_up_onfly_FB: ARRAY[0..7] OF INT;
	array_dest_up_onfly_FB: ARRAY[0..7] OF INT;
	array_prio_up_stored_FB: ARRAY[0..7] OF INT;
	array_dest_up_stored_FB: ARRAY[0..7] OF INT;
	
	array_prio_down_onfly_FB: ARRAY[0..7] OF INT;
	array_dest_down_onfly_FB: ARRAY[0..7] OF INT;
	array_prio_down_stored_FB: ARRAY[0..7] OF INT;
	array_dest_down_stored_FB: ARRAY[0..7] OF INT;
	
END_VAR
VAR
//indici di scrittura degli array
	j: INT;
	j1: INT;
	h: INT;
	h1: INT;
// per riordinare gli array
	i: INT;
	k: INT;
	var1: INT;
	var2: INT;
//priorità
	prio: INT;
//per controllare se resettare gli indici di scrittura degli array
	cont_FB: INT;
	cont_up_fly: INT;
	cont_up_stored: INT;
	cont_down_fly: INT;
	cont_down_stored: INT;
END_VAR

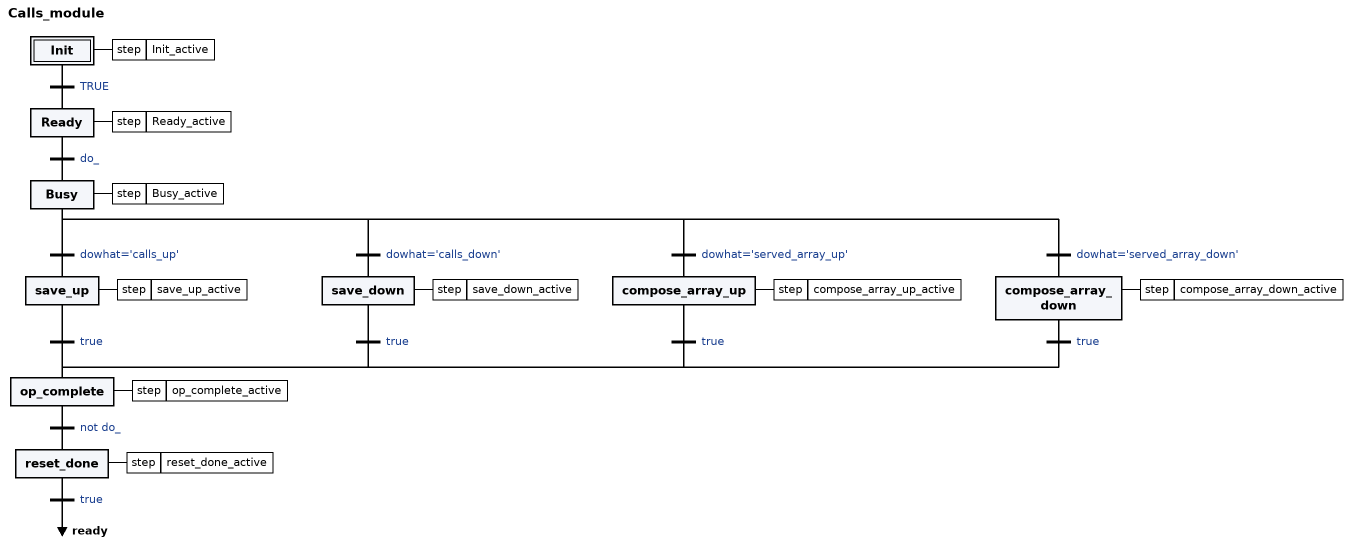
INITIAL_STEP Init:
    Init_active(N);  // step action
END_STEP
TRANSITION FROM Init TO Ready
    := TRUE;
END_TRANSITION
STEP Ready:
    Ready_active(N);  // step action
END_STEP
TRANSITION FROM Ready TO Busy
    := do_;
END_TRANSITION
STEP Busy:
    Busy_active(N);  // step action
END_STEP
TRANSITION FROM Busy TO save_up
    := dowhat='calls_up';
END_TRANSITION
STEP save_up:
    save_up_active(N);  // step action
END_STEP
TRANSITION FROM save_up TO op_complete
    := true;
END_TRANSITION
TRANSITION FROM Busy TO save_down
    := dowhat='calls_down';
END_TRANSITION
STEP save_down:
    save_down_active(N);  // step action
END_STEP
TRANSITION FROM save_down TO op_complete
    := true;
END_TRANSITION
TRANSITION FROM Busy TO compose_array_up
    := dowhat='served_array_up';
END_TRANSITION
STEP compose_array_up:
    compose_array_up_active(N);  // step action
END_STEP
TRANSITION FROM compose_array_up TO op_complete
    := true;
END_TRANSITION
TRANSITION FROM Busy TO compose_array_down
    := dowhat='served_array_down';
END_TRANSITION
STEP compose_array_down:
    compose_array_down_active(N);  // step action
END_STEP
TRANSITION FROM compose_array_down TO op_complete
    := true;
END_TRANSITION
STEP op_complete:
    op_complete_active(N);  // step action
END_STEP
TRANSITION FROM op_complete TO reset_done
    := not do_;
END_TRANSITION
STEP reset_done:
    reset_done_active(N);  // step action
END_STEP
TRANSITION FROM reset_done TO ready
    := true;
END_TRANSITION

ACTION Busy_active:
State:='busy';
END_ACTION

ACTION Ready_active:
State:='ready';
END_ACTION

ACTION op_complete_active:
//controllo se gli array posseggono otto elementi su otto a prio=8
cont_FB:=0;
WHILE cont_FB<8 DO
	IF array_prio_up_onfly_FB[cont_FB] = 8 THEN
		cont_up_fly:=cont_up_fly+1;
	END_IF
	IF array_prio_up_stored_FB[cont_FB] = 8 THEN
		cont_up_stored:=cont_up_stored+1;
	END_IF
	IF array_prio_down_onfly_FB[cont_FB] = 8 THEN
		cont_down_fly:=cont_down_fly+1;
	END_IF
	IF array_prio_down_stored_FB[cont_FB] = 8 THEN
		cont_down_stored:=cont_down_stored+1;
	END_IF
END_WHILE

IF cont_up_fly=8 OR j=7 THEN
	j:=0;
END_IF

IF cont_up_stored=8 OR j1=7 THEN
	j1:=0;
END_IF

IF cont_down_fly=8 OR h=7 THEN
	h:=0;
END_IF

IF cont_down_stored=8 OR h1=7THEN
	h1:=0;
END_IF
cont_up_fly:=0;
cont_up_stored:=0;
cont_down_fly:=0;
cont_down_stored:=0;
done:=true;
END_ACTION

ACTION reset_done_active:
done:=FALSE;
END_ACTION

ACTION save_up_active:
//sono negli array delle chiamate up
	IF dest_floor_FB>curr_floor_FB THEN //vado negli array per le chiamate onfly
		prio:= dest_floor_FB-curr_floor_FB; // definisco la priorità
		array_prio_up_onfly_FB[j]:= prio; // carico nell'array delle prio
		array_dest_up_onfly_FB[j]:= dest_floor_FB; // carico nell'array delle dest
		j:=j+1; // incremento l'indice entro cui metterò la prossima chiamata verso l'alto 
		k:=0;
		i:=1;
		//PARTO CON L'ORDINAMENTO CON IL SELECTION SORTER
		WHILE i<8 DO
			var1:= array_prio_up_onfly_FB[i];
			var2:= array_dest_up_onfly_FB[i];
			k:=i-1;
			WHILE k>=0 AND array_prio_up_onfly_FB[k]>var1 DO
				array_prio_up_onfly_FB[k+1]:= array_prio_up_onfly_FB[k];
				array_dest_up_onfly_FB[k+1]:= array_dest_up_onfly_FB[k];
			END_WHILE
			array_prio_up_onfly_FB[k+1]:= var1;
			array_dest_up_onfly_FB[k+1]:= var2;
		END_WHILE
	ELSE //vado negli array per le chiamate stored
		prio:= curr_floor_FB-dest_floor_FB; // definisco la priorità
		array_prio_up_stored_FB[j1]:= prio; // carico nell'array delle prio
		array_dest_up_stored_FB[j1]:= dest_floor_FB; // carico nell'array delle dest
		j1:=j1+1; // incremento l'indice entro cui metterò la prossima chiamata verso l'alto 
		k:=0;
		i:=1;
		//PARTO CON L'ORDINAMENTO CON IL SELECTION SORTER
		WHILE i<8 DO
			var1:= array_prio_up_stored_FB[i];
			var2:= array_dest_up_stored_FB[i];
			k:=i-1;
			WHILE k>=0 AND array_prio_up_onfly_FB[k]>var1 DO
				array_prio_up_stored_FB[k+1]:= array_prio_up_stored_FB[k];
				array_dest_up_stored_FB[k+1]:=array_dest_up_stored_FB[k];
			END_WHILE
			array_prio_up_stored_FB[k+1]:= var1;
			array_dest_up_stored_FB[k+1]:= var2;
		END_WHILE
	END_IF
END_ACTION

ACTION Init_active:
j:=0;
j1:=0;
h:=0;
h1:=0;

WHILE j<8 DO 
	array_prio_up_onfly_FB[j]:=8;
	array_dest_up_onfly_FB[j]:=8;
	array_prio_up_stored_FB[j]:=8;
	array_dest_up_stored_FB[j]:=8;
	
	array_prio_down_onfly_FB[j]:=8;
	array_dest_down_onfly_FB[j]:=8;
	array_prio_down_stored_FB[j]:=8;
	array_dest_down_stored_FB[j]:=8;
END_WHILE
j:=0;
END_ACTION

ACTION save_down_active:
//ENTRO NEGLI ARRAY PER LE CHIAMATE VERSO IL BASSO
IF dest_floor_FB<curr_floor_FB THEN //vado negli array per le chiamate onfly
		prio:= curr_floor_FB-dest_floor_FB; // definisco la priorità
		array_prio_down_onfly_FB[h]:= prio; // carico nell'array delle prio
		array_dest_down_onfly_FB[h]:= dest_floor_FB; // carico nell'array delle dest
		h:=h+1; // incremento l'indice entro cui metterò la prossima chiamata verso l'alto 
		k:=0;
		i:=1;
		//PARTO CON L'ORDINAMENTO CON IL SELECTION SORTER
		WHILE i<8 DO
			var1:= array_prio_down_onfly_FB[i];
			var2:= array_dest_down_onfly_FB[i];
			k:=i-1;
			WHILE k>=0 AND array_prio_down_onfly_FB[k]>var1 DO
				array_prio_down_onfly_FB[k+1]:= array_prio_down_onfly_FB[k];
				array_dest_down_onfly_FB[k+1]:=array_dest_down_onfly_FB[k];
			END_WHILE
			array_prio_down_onfly_FB[k+1]:= var1;
			array_dest_down_onfly_FB[k+1]:= var2;
		END_WHILE
	ELSE //vado negli array per le chiamate stored
		prio:= curr_floor_FB-dest_floor_FB; // definisco la priorità
		array_prio_down_stored_FB[h1]:= prio; // carico nell'array delle prio
		array_dest_down_stored_FB[h1]:= dest_floor_FB; // carico nell'array delle dest
		h1:=h1+1; // incremento l'indice entro cui metterò la prossima chiamata verso l'alto 
		k:=0;
		i:=1;
		//PARTO CON L'ORDINAMENTO CON IL SELECTION SORTER
		WHILE i<8 DO
			var1:= array_prio_down_stored_FB[i];
			var2:= array_dest_down_stored_FB[i];
			k:=i-1;
			WHILE k>=0 AND array_prio_down_stored_FB[k]>var1 DO
				array_prio_down_stored_FB[k+1]:= array_prio_down_stored_FB[k];
				array_dest_down_stored_FB[k+1]:=array_dest_down_stored_FB[k];
			END_WHILE
			array_prio_down_stored_FB[k+1]:= var1;
			array_dest_down_stored_FB[k+1]:= var2;
		END_WHILE
	END_IF
END_ACTION

ACTION compose_array_up_active:
//quando la chiamata è stata servita, la faccio diventare di prio 8
array_prio_up_onfly_FB[0]:=8;
array_dest_up_onfly_FB[0]:=8;

//PARTO CON L'ORDINAMENTO CON IL SELECTION SORTER
k:=0;
i:=1;
WHILE i<8 DO
	var1:= array_prio_up_onfly_FB[i];
	var2:= array_dest_up_onfly_FB[i];
	k:=i-1;
	WHILE k>=0 AND array_prio_up_onfly_FB[k]>var1 DO
		array_prio_up_onfly_FB[k+1]:= array_prio_up_onfly_FB[k];
		array_dest_up_onfly_FB[k+1]:= array_dest_up_onfly_FB[k];
	END_WHILE
	array_prio_up_onfly_FB[k+1]:= var1;
	array_dest_up_onfly_FB[k+1]:= var2;
END_WHILE
END_ACTION

ACTION compose_array_down_active:
//quando la chiamata è stata servita, la faccio diventare di prio 8
array_prio_down_onfly_FB[0]:=8;
array_dest_down_onfly_FB[0]:=8;

//PARTO CON L'ORDINAMENTO CON IL SELECTION SORTER
k:=0;
i:=1;
WHILE i<8 DO
	var1:= array_prio_down_onfly_FB[i];
	var2:= array_dest_down_onfly_FB[i];
	k:=i-1;
	WHILE k>=0 AND array_prio_down_onfly_FB[k]>var1 DO
		array_prio_down_onfly_FB[k+1]:= array_prio_down_onfly_FB[k];
		array_dest_down_onfly_FB[k+1]:=array_dest_down_onfly_FB[k];
	END_WHILE
	array_prio_down_onfly_FB[k+1]:= var1;
	array_dest_down_onfly_FB[k+1]:= var2;
END_WHILE
END_ACTION

END_FUNCTION_BLOCK

// Device/Application/Policy
PROGRAM Policy
VAR
	sync: BOOL;
	Opok: BOOL;
END_VAR

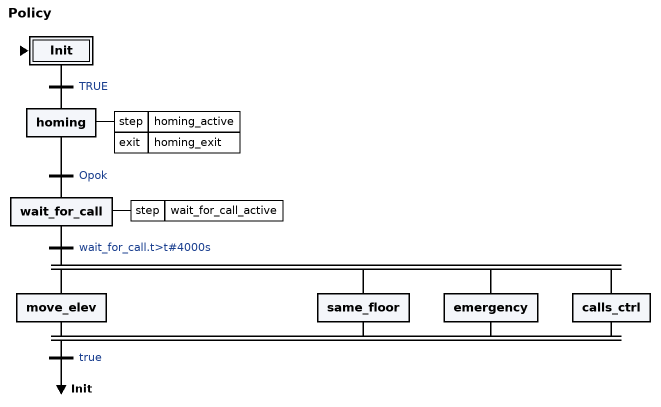
INITIAL_STEP Init:
END_STEP
TRANSITION FROM Init TO homing
    := TRUE;
END_TRANSITION
STEP homing:
    homing_active(N);  // step action
    homing_exit(P0);  // exit action
END_STEP
TRANSITION FROM homing TO wait_for_call
    := Opok;
END_TRANSITION
STEP wait_for_call:
    wait_for_call_active(N);  // step action
END_STEP
TRANSITION FROM wait_for_call TO (move_elev, same_floor, emergency, calls_ctrl)
    := wait_for_call.t>t#4000s;
END_TRANSITION
STEP move_elev:
END_STEP
STEP same_floor:
END_STEP
STEP emergency:
END_STEP
STEP calls_ctrl:
END_STEP
TRANSITION FROM (move_elev, same_floor, emergency, calls_ctrl) TO Init
    := true;
END_TRANSITION

ACTION homing_active:
//ATTUAZIONE DELLA FASE DI HOMING
IF Homing_Limit_module_0.State='Ready' THEN
	Homing_Limit_module_0.Do_:=TRUE;
	Homing_Limit_module_0.DoWhat:='homing';
END_IF

IF Homing_Limit_module_0.Done AND Homing_Limit_module_0.State='Busy' THEN
	Homing_Limit_module_0.Do_:=FALSE;
	sync:=TRUE;
END_IF

Opok:= sync AND NOT Homing_Limit_module_0.Done;

current := 0; //Aggiornamento del piano tramite il contatore
END_ACTION

ACTION homing_exit:
sync:=FALSE;
Opok:=FALSE;
END_ACTION

ACTION wait_for_call_active:
// IF Lights_module_0.State='Ready' THEN
// 	Lights_module_0.Start_:=TRUE;
// 	Lights_module_0.Stop:=FALSE;
// 	(*Temperature1.StartWhat:='Warm60';*)
// END_IF
END_ACTION

END_PROGRAM

// Device/Application/GAs/Serve_call_module
FUNCTION_BLOCK Serve_call_module
VAR_INPUT
	Start_: BOOL;
	Stop: BOOL;
	curr_floor_FB: INT;
	dest_floor_FB: INT;
	DeckSensor_FB: BOOL;
	RampSensor_FB: BOOL;
	RampSensor_target_FB: BOOL; // la policy calcolerà la dest_target 
END_VAR
VAR_OUTPUT
	state: STRING;
	up_flag_FB: BOOL;
END_VAR
VAR
	sync: BOOL;
	Opok: BOOL;

END_VAR

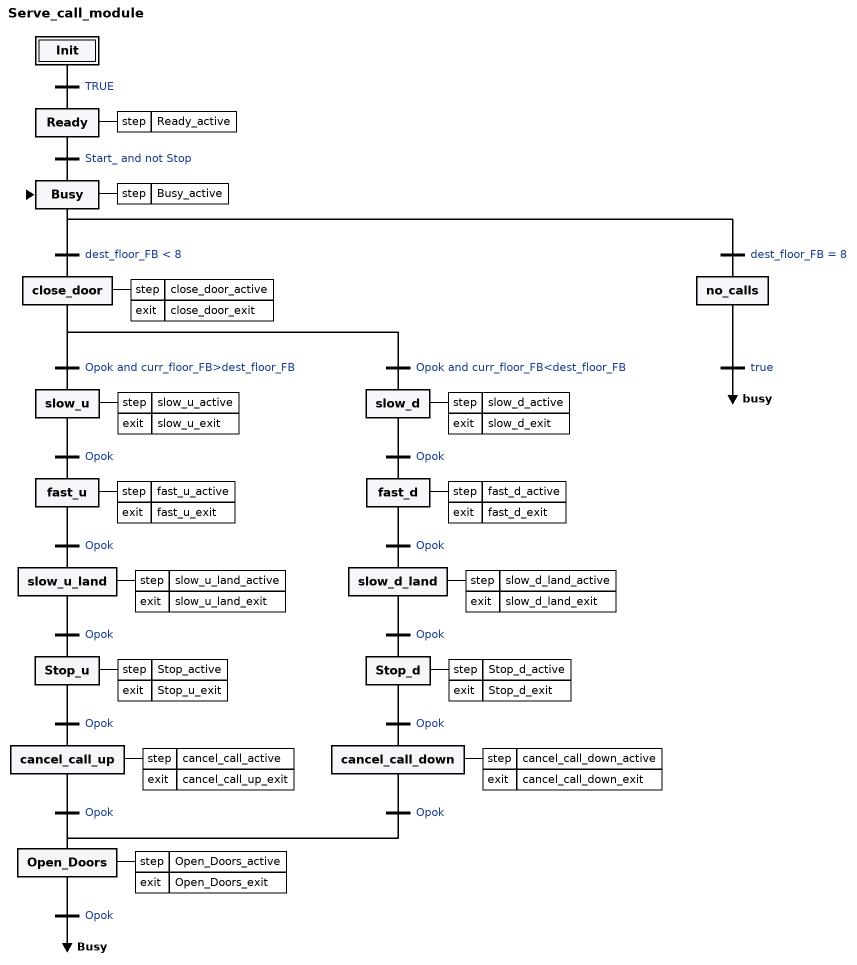
INITIAL_STEP Init:
END_STEP
TRANSITION FROM Init TO Ready
    := TRUE;
END_TRANSITION
STEP Ready:
    Ready_active(N);  // step action
END_STEP
TRANSITION FROM Ready TO Busy
    := Start_ and not Stop;
END_TRANSITION
STEP Busy:
    Busy_active(N);  // step action
END_STEP
TRANSITION FROM Busy TO close_door
    := dest_floor_FB < 8;
END_TRANSITION
STEP close_door:
    close_door_active(N);  // step action
    close_door_exit(P0);  // exit action
END_STEP
TRANSITION FROM close_door TO slow_u
    := Opok and curr_floor_FB>dest_floor_FB;
END_TRANSITION
STEP slow_u:
    slow_u_active(N);  // step action
    slow_u_exit(P0);  // exit action
END_STEP
TRANSITION FROM slow_u TO fast_u
    := Opok;
END_TRANSITION
STEP fast_u:
    fast_u_active(N);  // step action
    fast_u_exit(P0);  // exit action
END_STEP
TRANSITION FROM fast_u TO slow_u_land
    := Opok;
END_TRANSITION
STEP slow_u_land:
    slow_u_land_active(N);  // step action
    slow_u_land_exit(P0);  // exit action
END_STEP
TRANSITION FROM slow_u_land TO Stop_u
    := Opok;
END_TRANSITION
STEP Stop_u:
    Stop_active(N);  // step action
    Stop_u_exit(P0);  // exit action
END_STEP
TRANSITION FROM Stop_u TO cancel_call_up
    := Opok;
END_TRANSITION
STEP cancel_call_up:
    cancel_call_active(N);  // step action
    cancel_call_up_exit(P0);  // exit action
END_STEP
TRANSITION FROM cancel_call_up TO Open_Doors
    := Opok;
END_TRANSITION
TRANSITION FROM close_door TO slow_d
    := Opok and curr_floor_FB<dest_floor_FB;
END_TRANSITION
STEP slow_d:
    slow_d_active(N);  // step action
    slow_d_exit(P0);  // exit action
END_STEP
TRANSITION FROM slow_d TO fast_d
    := Opok;
END_TRANSITION
STEP fast_d:
    fast_d_active(N);  // step action
    fast_d_exit(P0);  // exit action
END_STEP
TRANSITION FROM fast_d TO slow_d_land
    := Opok;
END_TRANSITION
STEP slow_d_land:
    slow_d_land_active(N);  // step action
    slow_d_land_exit(P0);  // exit action
END_STEP
TRANSITION FROM slow_d_land TO Stop_d
    := Opok;
END_TRANSITION
STEP Stop_d:
    Stop_d_active(N);  // step action
    Stop_d_exit(P0);  // exit action
END_STEP
TRANSITION FROM Stop_d TO cancel_call_down
    := Opok;
END_TRANSITION
STEP cancel_call_down:
    cancel_call_down_active(N);  // step action
    cancel_call_down_exit(P0);  // exit action
END_STEP
TRANSITION FROM cancel_call_down TO Open_Doors
    := Opok;
END_TRANSITION
TRANSITION FROM Busy TO no_calls
    := dest_floor_FB = 8;
END_TRANSITION
STEP no_calls:
END_STEP
TRANSITION FROM no_calls TO busy
    := true;
END_TRANSITION
STEP Open_Doors:
    Open_Doors_active(N);  // step action
    Open_Doors_exit(P0);  // exit action
END_STEP
TRANSITION FROM Open_Doors TO Busy
    := Opok;
END_TRANSITION

ACTION Ready_active:
State:='ready';
END_ACTION

ACTION Busy_active:
State:='busy';
END_ACTION

ACTION close_door_exit:
sync:=FALSE;
Opok:=FALSE;
END_ACTION

ACTION slow_d_active:
//VERSO IL BASSO LENTO
IF Dir_Vel_module_0.State='Ready' THEN
	Dir_Vel_module_0.Do_:=TRUE;
	Dir_Vel_module_0.DoWhat:='slow_mode';
	up_flag_FB:=FALSE;
END_IF

IF Dir_Vel_module_0.Done AND Dir_Vel_module_0.State='Busy' AND NOT RampSensor_FB THEN
	Dir_Vel_module_0.Do_:=FALSE;
	sync:=TRUE;
END_IF

Opok:= sync AND NOT Dir_Vel_module_0.Done;
END_ACTION

ACTION slow_d_exit:
sync:=FALSE;
Opok:=FALSE;
END_ACTION

ACTION close_door_active:
//CHIUSURA PORTE 
IF door_module_0.State='Ready' THEN
	door_module_0.Do_:=TRUE;
	door_module_0.DoWhat:='close_door';
END_IF

IF door_module_0.Done AND door_module_0.State='Busy' THEN
	door_module_0.Do_:=FALSE;
	sync:=TRUE;
END_IF

Opok:= sync and not door_module_0.Done;
END_ACTION

ACTION slow_u_active:
//VERSO L'ALTO LENTO
IF Dir_Vel_module_0.State='Ready' THEN
	Dir_Vel_module_0.Do_:=TRUE;
	Dir_Vel_module_0.DoWhat:='slow_mode';
	up_flag_FB:=TRUE;
END_IF

IF Dir_Vel_module_0.Done AND Dir_Vel_module_0.State='Busy' AND NOT RampSensor_FB THEN
	Dir_Vel_module_0.Do_:=FALSE;
	sync:=TRUE;
END_IF

Opok:= sync AND NOT Dir_Vel_module_0.Done;
END_ACTION

ACTION fast_u_active:
//VERSO L'ALTO VELOCE
IF Dir_Vel_module_0.State='Ready' THEN
	Dir_Vel_module_0.Do_:=TRUE;
	Dir_Vel_module_0.DoWhat:='fast_mode';
	up_flag_FB:=TRUE;
END_IF

IF Dir_Vel_module_0.Done AND Dir_Vel_module_0.State='Busy' AND RampSensor_target_FB THEN
	Dir_Vel_module_0.Do_:=FALSE;
	sync:=TRUE;
END_IF

Opok:= sync AND NOT Dir_Vel_module_0.Done;
END_ACTION

ACTION slow_u_land_active:
//VERSO L'ALTO LENTO
IF Dir_Vel_module_0.State='Ready' THEN
	Dir_Vel_module_0.Do_:=TRUE;
	Dir_Vel_module_0.DoWhat:='slow_mode';
	up_flag_FB:=TRUE;
END_IF

IF Dir_Vel_module_0.Done AND Dir_Vel_module_0.State='Busy' AND DeckSensor_FB THEN
	Dir_Vel_module_0.Do_:=FALSE;
	sync:=TRUE;
END_IF

Opok:= sync AND NOT Dir_Vel_module_0.Done;
END_ACTION

ACTION Stop_active:
//STOP
IF Dir_Vel_module_0.State='Ready' THEN
	Dir_Vel_module_0.Do_:=TRUE;
	Dir_Vel_module_0.DoWhat:='stop_mode';
END_IF

IF Dir_Vel_module_0.Done AND Dir_Vel_module_0.State='Busy' THEN
	Dir_Vel_module_0.Do_:=FALSE;
	sync:=TRUE;
END_IF

Opok:= sync AND NOT Dir_Vel_module_0.Done;
END_ACTION

ACTION Open_Doors_active:
//APERTURA PORTE 
IF door_module_0.State='Ready' THEN
	door_module_0.Do_:=TRUE;
	door_module_0.DoWhat:='open_door';
END_IF

IF door_module_0.Done AND door_module_0.State='Busy' THEN
	door_module_0.Do_:=FALSE;
	sync:=TRUE;
END_IF

Opok:= sync AND NOT door_module_0.Done;
END_ACTION

ACTION slow_u_exit:
sync:=FALSE;
Opok:=FALSE;
END_ACTION

ACTION fast_u_exit:
sync:=FALSE;
Opok:=FALSE;
END_ACTION

ACTION slow_u_land_exit:
sync:=FALSE;
Opok:=FALSE;
END_ACTION

ACTION Stop_u_exit:
sync:=FALSE;
Opok:=FALSE;
END_ACTION

ACTION Open_Doors_exit:
sync:=FALSE;
Opok:=FALSE;
END_ACTION

ACTION fast_d_active:
//VERSO IL BASSO VELOCE
IF Dir_Vel_module_0.State='Ready' THEN
	Dir_Vel_module_0.Do_:=TRUE;
	Dir_Vel_module_0.DoWhat:='fast_mode';
	up_flag_FB:=FALSE;
END_IF

IF Dir_Vel_module_0.Done AND Dir_Vel_module_0.State='Busy' AND RampSensor_target_FB THEN
	Dir_Vel_module_0.Do_:=FALSE;
	sync:=TRUE;
END_IF

Opok:= sync AND NOT Dir_Vel_module_0.Done;
END_ACTION

ACTION slow_d_land_active:
//VERSO IL BASSO LENTO
IF Dir_Vel_module_0.State='Ready' THEN
	Dir_Vel_module_0.Do_:=TRUE;
	Dir_Vel_module_0.DoWhat:='slow_mode';
	up_flag_FB:=FALSE;
END_IF

IF Dir_Vel_module_0.Done AND Dir_Vel_module_0.State='Busy' AND DeckSensor_FB THEN
	Dir_Vel_module_0.Do_:=FALSE;
	sync:=TRUE;
END_IF

Opok:= sync AND NOT Dir_Vel_module_0.Done;
END_ACTION

ACTION Stop_d_active:
//STOP
IF Dir_Vel_module_0.State='Ready' THEN
	Dir_Vel_module_0.Do_:=TRUE;
	Dir_Vel_module_0.DoWhat:='stop_mode';
END_IF

IF Dir_Vel_module_0.Done AND Dir_Vel_module_0.State='Busy' THEN
	Dir_Vel_module_0.Do_:=FALSE;
	sync:=TRUE;
END_IF

Opok:= sync AND NOT Dir_Vel_module_0.Done;
END_ACTION

ACTION fast_d_exit:
sync:=FALSE;
Opok:=FALSE;
END_ACTION

ACTION slow_d_land_exit:
sync:=FALSE;
Opok:=FALSE;
END_ACTION

ACTION Stop_d_exit:
sync:=FALSE;
Opok:=FALSE;
END_ACTION

ACTION cancel_call_active:
// UTILIZZO IL COMANDO PER CANCELLARE LA CHIAMATA APPENA SERVITA
IF Dir_Vel_module_0.State='Ready' THEN
	Dir_Vel_module_0.Do_:=TRUE;
	Dir_Vel_module_0.DoWhat:='served_array_up';
END_IF

IF Dir_Vel_module_0.Done AND Dir_Vel_module_0.State='Busy' THEN
	Dir_Vel_module_0.Do_:=FALSE;
	sync:=TRUE;
END_IF

Opok:= sync AND NOT Dir_Vel_module_0.Done;
END_ACTION

ACTION cancel_call_down_active:
// UTILIZZO IL COMANDO PER CANCELLARE LA CHIAMATA APPENA SERVITA
IF Dir_Vel_module_0.State='Ready' THEN
	Dir_Vel_module_0.Do_:=TRUE;
	Dir_Vel_module_0.DoWhat:='served_array_down';
END_IF

IF Dir_Vel_module_0.Done AND Dir_Vel_module_0.State='Busy' THEN
	Dir_Vel_module_0.Do_:=FALSE;
	sync:=TRUE;
END_IF

Opok:= sync AND NOT Dir_Vel_module_0.Done;
END_ACTION

ACTION cancel_call_up_exit:
sync:=FALSE;
Opok:=FALSE;
END_ACTION

ACTION cancel_call_down_exit:
sync:=FALSE;
Opok:=FALSE;
END_ACTION

END_FUNCTION_BLOCK

// Device/Application/Visualization
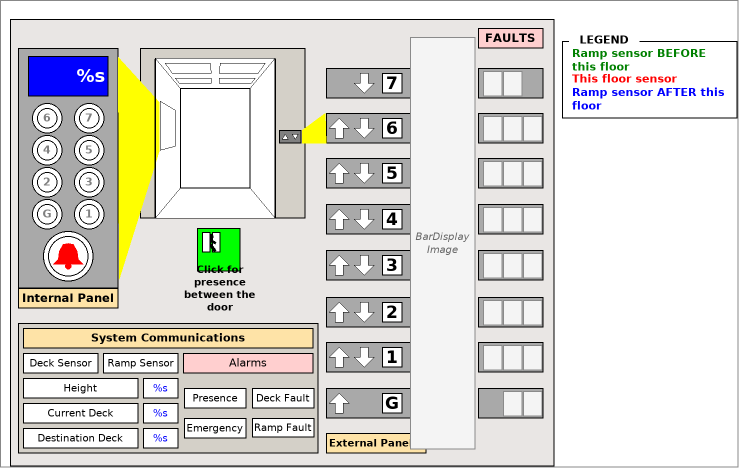
VISUALIZATION Visualization  // 739x468
    Rectangle (10,19 544x447)
    Rectangle (197,228 43x43), colour toggle: GVL.Presence
    Rectangle (18,323 300x130)
    Rectangle (326,433 100x20), "External Panels"
    Rectangle (326,342 100x30)
    Rectangle (382,347 20x20), "1"
    Polygon (354,357) (360,357) (360,347) (368,347) (368,357) (374,357) (364,367), colour toggle: GVL.DownDeck1Vis
        tap GVL.DownDeck1
    Polygon (329,357) (335,357) (335,367) (343,367) (343,357) (349,357) (339,347), colour toggle: GVL.UpDeck1Vis
        tap GVL.UpDeck1
    Rectangle (326,297 100x30)
    Rectangle (382,302 20x20), "2"
    Polygon (354,312) (360,312) (360,302) (368,302) (368,312) (374,312) (364,322), colour toggle: GVL.DownDeck2Vis
        tap GVL.DownDeck2
    Polygon (329,312) (335,312) (335,322) (343,322) (343,312) (349,312) (339,302), colour toggle: GVL.UpDeck2Vis
        tap GVL.UpDeck2
    Rectangle (326,250 100x30)
    Rectangle (382,255 20x20), "3"
    Polygon (354,265) (360,265) (360,255) (368,255) (368,265) (374,265) (364,275), colour toggle: GVL.DownDeck3Vis
        tap GVL.DownDeck3
    Polygon (329,265) (335,265) (335,275) (343,275) (343,265) (349,265) (339,255), colour toggle: GVL.UpDeck3Vis
        tap GVL.UpDeck3
    Rectangle (326,204 100x30)
    Rectangle (382,209 20x20), "4"
    Polygon (354,219) (360,219) (360,209) (368,209) (368,219) (374,219) (364,229), colour toggle: GVL.DownDeck4Vis
        tap GVL.DownDeck4
    Polygon (329,219) (335,219) (335,229) (343,229) (343,219) (349,219) (339,209), colour toggle: GVL.UpDeck4Vis
        tap GVL.UpDeck4
    Rectangle (326,158 100x30)
    Rectangle (382,163 20x20), "5"
    Polygon (354,173) (360,173) (360,163) (368,163) (368,173) (374,173) (364,183), colour toggle: GVL.DownDeck5Vis
        tap GVL.DownDeck5
    Polygon (329,173) (335,173) (335,183) (343,183) (343,173) (349,173) (339,163), colour toggle: GVL.UpDeck5Vis
        tap GVL.UpDeck5
    Rectangle (326,113 100x30)
    Rectangle (382,118 20x20), "6"
    Polygon (354,128) (360,128) (360,118) (368,118) (368,128) (374,128) (364,138), colour toggle: GVL.DownDeck6Vis
        tap GVL.DownDeck6
    Polygon (329,128) (335,128) (335,138) (343,138) (343,128) (349,128) (339,118), colour toggle: GVL.UpDeck6Vis
        tap GVL.UpDeck6
    Rectangle (326,68 100x30)
    Rectangle (382,73 20x20), "7"
    Polygon (354,83) (360,83) (360,73) (368,73) (368,83) (374,83) (364,93), colour toggle: GVL.DownDeck7Vis
        tap GVL.DownDeck7
    Rectangle (326,388 100x30)
    Rectangle (382,393 20x20), "G"
    Polygon (329,403) (335,403) (335,413) (343,413) (343,403) (349,403) (339,393), colour toggle: GVL.UpDeckGVis
        tap GVL.UpDeckG
    RoundedRectangle (18,48 100x240)
    Rectangle (18,288 100x20), "Internal Panel"
    Ellipse (74,199 30x30), colour toggle: GVL.P1Vis
    Ellipse (79,204 20x20), "1"
        tap GVL.P1
    Ellipse (32,199 30x30), colour toggle: GVL.PGVis
    Ellipse (37,204 20x20), "G"
        tap GVL.PG
    Ellipse (74,167 30x30), colour toggle: GVL.P3Vis
    Ellipse (79,172 20x20), "3"
        tap GVL.P3
    Ellipse (32,167 30x30), colour toggle: GVL.P2Vis
    Ellipse (37,172 20x20), "2"
        tap GVL.P2
    Ellipse (74,135 30x30), colour toggle: GVL.P5Vis
    Ellipse (79,140 20x20), "5"
        tap GVL.P5
    Ellipse (32,135 30x30), colour toggle: GVL.P4Vis
    Ellipse (37,140 20x20), "4"
        tap GVL.P4
    Ellipse (74,103 30x30), colour toggle: GVL.P7Vis
    Ellipse (79,108 20x20), "7"
        tap GVL.P7
    Ellipse (32,103 30x30), colour toggle: GVL.P6Vis
    Ellipse (37,108 20x20), "6"
        tap GVL.P6
    Rectangle (28,56 80x40), "%s", text variable: GVL.Destination
    Ellipse (43,231 50x50), tooltip "EMERGENCY", colour toggle: GVL.Emergency
    Group (48,236 40x40)
        toggle GVL.Emergency
        Ellipse (0,0 40x40), tooltip "EMERGENCY"
        Polygon (5,28) (10,23) (11,15) (15,8) (20,7) (25,8) (29,15) (30,23) (35,28)
        Ellipse (17,27 6x6)
    Polygon (35,72) (45,62) (55,72), colour toggle: GVL.Motor_on AND GVL.Up
    Polygon (35,80) (45,90) (55,80), colour toggle: GVL.Motor_on AND NOT GVL.Up
    Group (140,48 165x170)
        Rectangle (0,0 165x170)
        Rectangle (15,10 120x160)
        Polygon (40,40) (15,10) (135,10) (110,40)
        Rectangle (40,40 70x100)
        Polygon (15,170) (40,140) (110,140) (135,170)
        Polygon (20,102) (20,53) (35,62) (35,98)
        Polygon (79,35) (79,30) (115,30) (111,35)
        Polygon (39,35) (35,30) (71,30) (71,35)
        Polygon (32,25) (25,15) (70,15) (71,25)
        Polygon (79,25) (80,15) (125,15) (118,25)
        Group (139,82 22x13)
            Rectangle (0,0 22x13)
            Polygon (3,9) (6,4) (9,9)
            Polygon (13,4) (16,9) (19,4)
    BarDisplayImage (410,37 65x412), value: GVL.Height, style: BarDisplayImage-Gray, scale format: %.0f, scale -20..160
        p3451962224: VisuNativeControl.IP_Offline.Browser
    Rectangle (478,68 65x30)
    Rectangle (478,342 65x30)
    Rectangle (478,297 65x30)
    Rectangle (478,250 65x30)
    Rectangle (478,204 65x30)
    Rectangle (478,158 65x30)
    Rectangle (478,113 65x30)
    Rectangle (478,388 65x30)
    RockerSwitch (483,345 19x25), variable: GVL.Ramp1Down, behaviour: TOGGLE, style: Switch-RockerSwitch-Green
    RockerSwitch (503,345 19x25), variable: GVL.Sensor1, behaviour: TOGGLE, style: Switch-RockerSwitch-Red
    RockerSwitch (523,345 19x25), variable: GVL.Ramp1Up, behaviour: TOGGLE, style: Switch-RockerSwitch-Blue
    RockerSwitch (483,300 19x25), variable: GVL.Ramp2Down, behaviour: TOGGLE, style: Switch-RockerSwitch-Green
    RockerSwitch (503,300 19x25), variable: GVL.Sensor2, behaviour: TOGGLE, style: Switch-RockerSwitch-Red
    RockerSwitch (523,300 19x25), variable: GVL.Ramp2Up, behaviour: TOGGLE, style: Switch-RockerSwitch-Blue
    RockerSwitch (483,253 19x25), variable: GVL.Ramp3Down, behaviour: TOGGLE, style: Switch-RockerSwitch-Green
    RockerSwitch (503,253 19x25), variable: GVL.Sensor3, behaviour: TOGGLE, style: Switch-RockerSwitch-Red
    RockerSwitch (523,253 19x25), variable: GVL.Ramp3Up, behaviour: TOGGLE, style: Switch-RockerSwitch-Blue
    RockerSwitch (483,207 19x25), variable: GVL.Ramp4Down, behaviour: TOGGLE, style: Switch-RockerSwitch-Green
    RockerSwitch (503,207 19x25), variable: GVL.Sensor4, behaviour: TOGGLE, style: Switch-RockerSwitch-Red
    RockerSwitch (523,207 19x25), variable: GVL.Ramp4Up, behaviour: TOGGLE, style: Switch-RockerSwitch-Blue
    RockerSwitch (483,161 19x25), variable: GVL.Ramp5Down, behaviour: TOGGLE, style: Switch-RockerSwitch-Green
    RockerSwitch (503,161 19x25), variable: GVL.Sensor5, behaviour: TOGGLE, style: Switch-RockerSwitch-Red
    RockerSwitch (523,161 19x25), variable: GVL.Ramp5Up, behaviour: TOGGLE, style: Switch-RockerSwitch-Blue
    RockerSwitch (483,116 19x25), variable: GVL.Ramp6Down, behaviour: TOGGLE, style: Switch-RockerSwitch-Green
    RockerSwitch (503,116 19x25), variable: GVL.Sensor6, behaviour: TOGGLE, style: Switch-RockerSwitch-Red
    RockerSwitch (523,116 19x25), variable: GVL.Ramp6Up, behaviour: TOGGLE, style: Switch-RockerSwitch-Blue
    RockerSwitch (483,71 19x25), variable: GVL.Ramp7Down, behaviour: TOGGLE, style: Switch-RockerSwitch-Green
    RockerSwitch (503,71 19x25), variable: GVL.Sensor7, behaviour: TOGGLE, style: Switch-RockerSwitch-Red
    RockerSwitch (503,391 19x25), variable: GVL.SensorG, behaviour: TOGGLE, style: Switch-RockerSwitch-Red
    RockerSwitch (523,391 19x25), variable: GVL.RampGUp, behaviour: TOGGLE, style: Switch-RockerSwitch-Blue
    Rectangle (478,28 65x20), "FAULTS"
    Polygon (302,130) (325,113) (326,143) (302,143), invisible if: (GVL.Closing OR GVL.Opening) OR GVL.Closed
    Polygon (118,57) (159,102) (159,151) (119,279), invisible if: (GVL.Closing OR GVL.Opening) OR GVL.Closed
    Rectangle (155,58 0x160)
        p3528305787: GVL.Door
    Rectangle (275,58 0x160)
        p3528305787: -GVL.Door
    Rectangle (23,328 290x20), "System Communications"
    Rectangle (183,353 130x20), "Alarms"
    Rectangle (23,353 75x20), "Deck Sensor", colour toggle: GVL.DeckSensor
    Rectangle (143,378 35x20), "%s", text variable: GVL.Height
    Rectangle (184,388 62x20), "Presence", colour toggle: GVL.Presence
    Rectangle (103,353 75x20), "Ramp Sensor", colour toggle: GVL.RampSensor
    Rectangle (143,403 35x20), "%s", text variable: GVL.Current
    Rectangle (143,428 35x20), "%s", text variable: GVL.Destination
    Rectangle (252,388 62x20), "Deck Fault", colour toggle: GVL.FaultSensorAlarm
    Rectangle (184,418 62x20), "Emergency", colour toggle: GVL.EmergencyVis
    Rectangle (252,418 62x19), "Ramp Fault", colour toggle: GVL.FaultRampAlarm
    Rectangle (23,378 115x20), "Height"
    Rectangle (23,403 115x20), "Current Deck"
    Rectangle (23,428 115x20), "Destination Deck"
    Group (562,25 175x93)
        Rectangle (0,16 175x77)
        Rectangle (7,39 160x30), "This floor sensor"
        Rectangle (7,59 160x30), "Ramp sensor AFTER this floor"
        Rectangle (7,0 70x30), "LEGEND"
        Rectangle (7,20 160x30), "Ramp sensor BEFORE this floor"
    Group (202,232 33x34)
        toggle GVL.Presence
        Rectangle (10,0 8x20)
        Polygon (5,10) (12,20) (14,18) (5,6)
        Ellipse (6,2 5x5)
        Polygon (4,8) (13,12) (14,10) (4,4)
        Rectangle (0,0 8x20)
    Rectangle (169,273 102x31), "Click for presence between the door"
END_VISUALIZATION
